FUNCTION_BLOCK ExecuteCylinder
VAR_INPUT
	ptBlock : POINTER TO CylinderBlockBase;
	Command : eCylinderCommands;
END_VAR
VAR_OUTPUT
	bDone : BOOL ;
END_VAR
VAR
END_VAR

// store command
ptBlock^.COMMAND_CACHED := Command;

bDone := ptBlock^.BIT_DONE AND NOT ptBlock^.BIT_WARNING AND (ptBlock^.COMMAND_CACHED = ptBlock^.LAST_COMMAND);

//reset surpress
IF bDone THEN
	ptBlock^.BIT_WARN_SUPPRESS := FALSE;
END_IF

END_FUNCTION_BLOCK

(* stored: Version 1.1.0.1, ProductVersion 3.1.4020.12
   POU ExecuteCylinder: Id {11dec6ea-9e30-46a6-91c5-0fe02040b602}, SpecialFunc None *)
